FUNCTION SetupHardware : BOOL
VAR
	iWoodBunkSlot : WoodBunk;
	iChipboardSlot : Chipboard;
	
	slotsArr : ARRAY[1..GVL.maxQueue] OF STRING;
	
	i : INT;
	j : INT;
	
	temp : INT;
END_VAR

MEMSET(ADR(slotsArr), 0, SIZEOF(slotsArr));
FOR iWoodBunkSlot:=1 TO WoodBunk.size-1 BY 1 DO //init wood bunk magazine slots
	slotsArr[iWoodBunkSlot] := TO_STRING(iWoodBunkSlot);
END_FOR
magazineA21Left.setupSlots(slotsArr);
magazineA21Right.setupSlots(slotsArr);


MEMSET(ADR(slotsArr), 0, SIZEOF(slotsArr));
FOR iChipboardSlot:=1 TO Chipboard.size-1 BY 1 DO //init chipboard skid slots
	slotsArr[iChipboardSlot] := TO_STRING(iChipboardSlot);
END_FOR
skidA21Left.setupSlots(slotsArr);
skidA21Right.setupSlots(slotsArr);


FOR i:=1 TO GVL.maxQueue BY 1 DO //get wood bunk magazine availability from robot
	magazineA21Left.setOccupancy(i := i, occupancy := IntegerBitAccess( TO_ULINT(robot1.inputs[3]), TO_ULINT(i-1)) );
	skidA21Left.setOccupancy(i := i, occupancy := IntegerBitAccess( TO_ULINT(robot1.inputs[4]), TO_ULINT(i-1)) );
	
	magazineA21Right.setOccupancy(i := i, occupancy := IntegerBitAccess( TO_ULINT(robot2.inputs[3]), TO_ULINT(i-1)) );
	skidA21Right.setOccupancy(i := i, occupancy := IntegerBitAccess( TO_ULINT(robot2.inputs[4]), TO_ULINT(i-1)) );
END_FOR

//enable all drives
verticalDriveA21Left.bEnable := 
verticalDriveA21Right.bEnable := 
horizontalDriveA21Left.bEnable := 
horizontalDriveA21Right.bEnable := 
pistonA21Bottom.bEnable := 
TRUE;

END_FUNCTION

(* stored: Version 1.1.0.1, ProductVersion 3.1.4024.11
   POU SetupHardware: Id {ad70243f-26d6-4655-b24b-2a994d19bc18}, SpecialFunc None *)
